Fanuc KAREL source: ka00175.KL

-- PROVISIONAL review KL for V1013-1; original PC SHA256 6ec4af303be210d982891ac3617825ae7fe30177b317b735244d1599e1413973
-- Incomplete behavior may be omitted. Consult companion uncertainty JSON. Do not deploy.
PROGRAM KA00175
%NOLOCKGROUP
BEGIN
  -- UNRESOLVED_PC offsets 5-19; opcodes 22,22,1E
  -- UNRESOLVED_PC offsets 24-28; opcodes 7F
END KA00175
